{attribute 'pack_mode' := '1'}
TYPE ST_AddTrafficLightDataIn :
STRUCT
	sCellID						: STRING(30);
	sID							: STRING(30);
	iPath						: UINT;
	rPosition					: REAL;

END_STRUCT
END_TYPE

(* stored: Version 1.1.0.1, ProductVersion 3.1.4024.5
   DUT ST_AddTrafficLightDataIn: Id {7ffd15b2-9c5c-4a98-a2e2-4cf821e2fa35} *)
